// TwinCAT 3 PLC project main_program
// ProgramVersion: 3.1.4024.0
// libraries:
//   Tc2_MC2, * (Beckhoff Automation GmbH)
//   Tc2_Standard, * (Beckhoff Automation GmbH)
//   Tc2_System, * (Beckhoff Automation GmbH)
//   Tc3_Module, * (Beckhoff Automation GmbH)
// project tree:
//   DUTs/ E_BiaxialState.TcDUT (not stored), E_PlcSystemStatus.TcDUT (not stored), E_SafetyState.TcDUT (not stored), E_SyncPoint.TcDUT (not stored), ST_settings.TcDUT, ST_MoveCommand.TcDUT, ST_SystemStatus.TcDUT
//   GVLs/ GVL_Axis.TcGVL
//   / PlcTask.TcTTO
//   POUs/ fb_MovementController.TcPOU, fb_AxisStatusPublisher.TcPOU (not stored), fb_BiaxialCoordinator.TcPOU (not stored), fb_safety.TcPOU, fb_StatusBuffer.TcPOU, MAIN.TcPOU
// real-time tasks:
//   TASK PlcTask: cycle T#10ms, priority 20, ADS port 350
// motion (NC):
//   TASK NC-Task 1 SAF: cycle T#2ms, priority 4, ADS port 501
//   TASK NC-Task 1 SVB: cycle T#10ms, priority 8, ADS port 511
//   AXIS xAxis (id 1)
//     Dynamic: Acceleration=150, Deceleration=150, Jerk=225
//     Velo: RefSearch=2, RefSync=5, SlowManual=5, FastManual=10, Maximum=100
//     OtherSettings: AllowMotionCmdToSlave=true
//     encoder EncType=19
//       EncPara: ScaleFactorNumerator=2, ScaleFactorDenominator=1048576, MaxCount=#xffffffff
//         SoftEndMaxControl: Range=10000
//         Inc: RefSearchInverse=true, RefPosition=-5
//     drive DrvType=16
//       DrvPara: MaxCount=#xffffffff, DriveControlDWord=#x00020100
//         Analog: TorqueSetpointScale=10, ScaleFactorActTorque=0.1
//         TimeComp: TaskDelayCycles=1
//     controller CtrType=1
//       CtrPara: PriorControlFactor=1
//         Observer: BandWidth=20
//   AXIS yAxis (id 2)
//     Dynamic: Acceleration=150, Deceleration=150, Jerk=225
//     Velo: RefSearch=2, RefSync=5, SlowManual=5, FastManual=10, Maximum=100
//     OtherSettings: AllowMotionCmdToSlave=true
//     encoder EncType=19
//       EncPara: ScaleFactorNumerator=2, ScaleFactorDenominator=1048576, MaxCount=#xffffffff
//         SoftEndMinControl: Enable=true
//         SoftEndMaxControl: Range=10000
//         Inc: RefSearchInverse=true, RefPosition=-5, RefMode=1
//     drive DrvType=16
//       DrvPara: MaxCount=#xffffffff, DriveControlDWord=#x00020100
//         Analog: TorqueSetpointScale=10, ScaleFactorActTorque=0.1
//         TimeComp: TaskDelayCycles=1
//     controller CtrType=1
//       CtrPara: PriorControlFactor=1
//         Observer: BandWidth=20
// I/O:
//   DEVICE Device 1 (EtherCAT), AmsNetId 5.85.113.174.2.1
//     Term 1 (EK1200) [EK1200-5000 EtherCAT Power supply (2A E-Bus)]
//       Term 2 (EL7062) [EL7062-0000 2Ch. Stepper motor output stage (48V, 3A)]
//       Term 3 (EL9510) [EL9510 Power supply terminal 10V]
//       Term 4 (EL3356-0020) [EL3356-0020 1Ch. Ana. Input Resistor Bridge Terminal, 24bit, High Precision, with calibration certificate]
//       Term 5 (EL3356-0020) [EL3356-0020 1Ch. Ana. Input Resistor Bridge Terminal, 24bit, High Precision, with calibration certificate]
//       Term 6 (EL9011) [EL9011 End Terminal]
// variable links:
//   NC-Task 1 SAF/Axes/xAxis <-> Device 1 (EtherCAT)/Term 1 (EK1200)/Term 2 (EL7062)
//     Drive/Inputs/In/nDataIn1 <-> DRV Following error actual value Channel 2/Following error actual value
//     Drive/Inputs/In/nDcOutputTime <-> InfoData/DcOutputShift
//     Drive/Inputs/In/nState1 <-> DRV Statusword Channel 2/Statusword
//     Drive/Inputs/In/nState2 <-> DRV Statusword Channel 2/Statusword @bit 8
//     Drive/Inputs/In/nState4 @bit 1 <-> WcState/InputToggle
//     Drive/Inputs/In/nState4 <-> WcState/WcState
//     Drive/Outputs/Out/nCtrl1 <-> DRV Controlword Channel 2/Controlword
//     Drive/Outputs/Out/nCtrl2 <-> DRV Controlword Channel 2/Controlword @bit 8
//     Drive/Outputs/Out/nDataOut1 <-> DRV Target position Channel 2/Target position
//     Enc/Inputs/In/nDataIn1 <-> FB Position Channel 2/Position
//     Enc/Inputs/In/nDcInputTime <-> InfoData/DcInputShift
//     Enc/Inputs/In/nState4 @bit 1 <-> WcState/InputToggle
//     Enc/Inputs/In/nState4 <-> WcState/WcState
//   NC-Task 1 SAF/Axes/yAxis <-> Device 1 (EtherCAT)/Term 1 (EK1200)/Term 2 (EL7062)
//     Drive/Inputs/In/nDataIn1 <-> DRV Following error actual value Channel 1/Following error actual value
//     Drive/Inputs/In/nDcOutputTime <-> InfoData/DcOutputShift
//     Drive/Inputs/In/nState1 <-> DRV Statusword Channel 1/Statusword
//     Drive/Inputs/In/nState2 <-> DRV Statusword Channel 1/Statusword @bit 8
//     Drive/Inputs/In/nState4 @bit 1 <-> WcState/InputToggle
//     Drive/Inputs/In/nState4 <-> WcState/WcState
//     Drive/Outputs/Out/nCtrl1 <-> DRV Controlword Channel 1/Controlword
//     Drive/Outputs/Out/nCtrl2 <-> DRV Controlword Channel 1/Controlword @bit 8
//     Drive/Outputs/Out/nDataOut1 <-> DRV Target position Channel 1/Target position
//     Enc/Inputs/In/nDataIn1 <-> FB Position Channel 1/Position
//     Enc/Inputs/In/nDcInputTime <-> InfoData/DcInputShift
//     Enc/Inputs/In/nState4 @bit 1 <-> WcState/InputToggle
//     Enc/Inputs/In/nState4 <-> WcState/WcState
//   main program/main program Instance <-> Device 1 (EtherCAT)/Term 1 (EK1200)/Term 2 (EL7062)
//     PlcTask Inputs/MAIN.nEndStopHx <-> DI Inputs Channel 2/Input 1
//     PlcTask Inputs/MAIN.nEndStopHy <-> DI Inputs Channel 1/Input 2
//     PlcTask Inputs/MAIN.nEndStopLx <-> DI Inputs Channel 1/Input 1
//     PlcTask Inputs/MAIN.nEndStopLy <-> DI Inputs Channel 2/Input 2
//   main program/main program Instance <-> Device 1 (EtherCAT)/Term 1 (EK1200)/Term 4 (EL3356-0020)
//     PlcTask Inputs/MAIN.nRawTenzoX <-> RMB Value (INT32)/Value
//   main program/main program Instance <-> Device 1 (EtherCAT)/Term 1 (EK1200)/Term 5 (EL3356-0020)
//     PlcTask Inputs/MAIN.nRawTenzoY <-> RMB Value (INT32)/Value
//   main program/main program Instance <-> NC-Task 1 SAF/Axes/xAxis
//     PlcTask Inputs/GVL_Axis.xAxis.NcToPlc <-> Outputs/ToPlc
//     PlcTask Outputs/GVL_Axis.xAxis.PlcToNc <-> Inputs/FromPlc
//   main program/main program Instance <-> NC-Task 1 SAF/Axes/yAxis
//     PlcTask Inputs/GVL_Axis.yAxis.NcToPlc <-> Outputs/ToPlc
//     PlcTask Outputs/GVL_Axis.yAxis.PlcToNc <-> Inputs/FromPlc

CONFIGURATION main_program
    RESOURCE PLC ON TwinCAT3
        TASK PlcTask(INTERVAL := T#10ms, PRIORITY := 20);
        PROGRAM MAIN WITH PlcTask : MAIN;
    END_RESOURCE
END_CONFIGURATION

// ---- DUTs/ST_settings.TcDUT
TYPE ST_Settings :
	STRUCT
		// Force-sensor calibration
		fTenzoCons   : LREAL := 0.01;
		fTenzoOffset : LREAL := 0.0;

		// Force control
		fKp : LREAL := 10;
		fKi : LREAL := 0.1;
		fIntegralLimit  : LREAL := 10;
		fForceTolerance : LREAL := 0.1;
		fMaxVelocity    : LREAL := 100;

		// Runtime force limit
		fMaxForce            : LREAL := 10;
		fForceReliefDistance : LREAL := 1.0; // fixed overforce release move [mm]
		fForceReliefVelocity : LREAL := 1.0; // release speed [mm/s]
	END_STRUCT
END_TYPE

// ---- DUTs/ST_MoveCommand.TcDUT
TYPE ST_MoveCommand :
	STRUCT
		// Mode 1: one relative move
		fMoveDistance : LREAL;
		fMoveVelocity : LREAL;

		// Mode 2: one PI-regulated force hold
		fTargetForce   : LREAL;
		fForceDuration : LREAL;
	
		// Command and service controls
		nMode       : INT;  // 1=relative move, 2=force/time, 3=test sequence
		bExecute    : BOOL; // Start movement
		bHalt       : BOOL; // Panic stop
		bPower      : BOOL; // Maintained motor-enable request
		bReset      : BOOL; // Reset errors
		bHome       : BOOL; // Start homing sequence
		bStartTar   : BOOL; // Start tare sequence
		bSavePosition : BOOL; // Capture the current axis position while idle
		bRestorePosition : BOOL; // Return to the saved coordinate while idle
		fRestoreVelocity : LREAL; // Saved-position return speed [mm/s]

		// Optional force pre-conditioning sequence
		bIncludePreTest : BOOL;
		bPreTestOnly    : BOOL;  // Run pre-test and post-test without a main test
		nPreCycleCount  : INT;   // Number of force load/unload cycles, 0..50
		bPreloadEnabled : BOOL;  // Apply one force preload before the first cycle
		fPreloadValue   : LREAL; // Signed preload force [N]
		fPreCycleLoadValue : LREAL; // Signed repeated preconditioning load target [N]
		fPreUnloadValue : LREAL; // Signed force unload target [N]
		bPreUnloadToStart : BOOL; // Return to sequence-start position instead of force unload
		fPreTestRate     : LREAL; // Positive motor speed magnitude [mm/s]
		fPreTestForceTolerance : LREAL := 0.1; // Force deadband for pre-test endpoints [N]
		fPreloadHoldTime : LREAL := 0.0; // Hold time for the initial preload endpoint [s]
		fPreCycleHoldTime : LREAL := 0.0; // Hold time for cyclic pre-conditioning endpoints [s]

		// Main test settings
		fTestRate      : LREAL; // Positive motor speed magnitude [mm/s]
		fSingleForceTolerance : LREAL := 0.1; // Force deadband for single-test endpoints [N]
		fSingleForceHoldTime : LREAL := 0.0; // Hold time for the single-test primary force endpoint [s]
		fCyclicForceTolerance : LREAL := 0.1; // Force deadband for cyclic endpoints [N]
		fCyclicForceHoldTime : LREAL := 0.0; // Hold time for cyclic force endpoints [s]

		// Test selection: >0=cyclic count, 0=single test
		nCycleCount : INT;
		nLoadMode   : INT;   // 1=displacement, 2=force
		fLoadValues : ARRAY[1..50] OF LREAL; // per-cycle level [mm] or signed force [N]
		nUnloadMode : INT;   // 1=displacement, 2=force
		fUnloadValues : ARRAY[1..50] OF LREAL; // per-cycle level [mm] or signed force [N]

		// Single test (nMode=3, nCycleCount=0); criterion 2 is optional OR
		nStop1Mode         : INT;   // 0=off, 1=displacement, 2=force
		fStop1Value        : LREAL;
		nStop2Mode         : INT;
		fStop2Value        : LREAL;

		// 0=stay, 1=saved position, 2=sequence start,
		// 3=pre-test final position, 4=unload to zero force
		nPostTestMode : INT;
	END_STRUCT
END_TYPE

// ---- DUTs/ST_SystemStatus.TcDUT
TYPE ST_SystemStatus :
	STRUCT
		fPosBuffer   : ARRAY[1..50] OF LREAL; // FIFO position data
		fTenzoBuffer : ARRAY[1..50] OF LREAL; // FIFO tenzo data
		nBufferHead  : INT := 50;             // Index of latest completely written sample
		nSampleCounter    : UDINT := 0;       // Monotonic counter for dropped-sample detection
		nOperationCounter : UDINT := 0;       // Incremented after each completed motion command
		nInterfaceVersion : UDINT := 5;       // MATLAB/PLC ADS contract version
		fTenzoTarOffset   : LREAL := 0.0;     // Calculated tar offset
		fActPosition : LREAL := 0.0;          // Absolute NC axis position
		
		bWorking     : BOOL;                   // PLC occupied; do not send a new test
		bTarWorking  : BOOL;                   // PLC is calculating tare
		bError       : BOOL;                   // Latched application or motion error
		nErrorCode   : UDINT := 0;             // Application error code (0 = no error)
		nAxisErrorID : UDINT := 0;             // Native TwinCAT/NC error ID
		bPowered     : BOOL;                   // Axis power is enabled
		bHoming      : BOOL;                   // Homing command is active
		bHomed       : BOOL;                   // NC axis reports a valid home reference
		bStopped     : BOOL;                   // Axis is at standstill
		bSavedPositionValid : BOOL;            // A return-to-saved reference is available
		nTestPhase   : BYTE := 0;              // 0 idle, 1 pretest, 2 test, 3 post-test
	END_STRUCT
END_TYPE

// ---- GVLs/GVL_Axis.TcGVL
VAR_GLOBAL
	// Axis handlers
	xAxis : Axis_REF;
	yAxis : Axis_REF;
END_VAR

// ---- POUs/MAIN.TcPOU
PROGRAM MAIN

VAR
	fbSafetyX : fb_safety;
	fbSafetyY : fb_safety;
	fbSystemBufferX : fb_StatusBuffer;
	fbSystemBufferY : fb_StatusBuffer;
	fbMovementControllerX : fb_MovementController;
	fbMovementControllerY : fb_MovementController;
	fbBiaxialCoordinator : fb_BiaxialCoordinator;
	fbStatusPublisherX : fb_AxisStatusPublisher;
	fbStatusPublisherY : fb_AxisStatusPublisher;
	
	// DUTs import
	stMoveCommandX : ST_MoveCommand;
	stMoveCommandY : ST_MoveCommand;

	stSystemStatusX : ST_SystemStatus;
	stSystemStatusY : ST_SystemStatus;

	stSettingsX : ST_Settings;
	stSettingsY : ST_Settings;

	// IO Links
    nRawTenzoX AT %I* : DINT;
	nRawTenzoY AT %I* : DINT;

	nEndStopLx AT %I* : BOOL;
	nEndStopHx AT %I* : BOOL;

	nEndStopLy AT %I* : BOOL;
	nEndStopHy AT %I* : BOOL;

	// Normalized physical limits: TRUE means that the switch is pressed.
	bEndStopLxActive : BOOL;
	bEndStopHxActive : BOOL;
	bEndStopLyActive : BOOL;
	bEndStopHyActive : BOOL;

	// PLC-owned synchronized start request
	bStartBiaxialTest : BOOL; // ADS one-shot after both axis commands are prepared

END_VAR

VAR_TEMP
	bBiaxialAxesReady : BOOL;
	bBiaxialCommonAbortRequest : BOOL;
END_VAR

////////////////////////////////
//////////   safety   //////////
////////////////////////////////

// Refresh NC status before making any safety or motion decision
GVL_Axis.xAxis.ReadStatus();
GVL_Axis.yAxis.ReadStatus();

// Normalize the active-low physical switches
bEndStopLxActive := NOT nEndStopLx;
bEndStopHxActive := NOT nEndStopHx;
bEndStopLyActive := NOT nEndStopLy;
bEndStopHyActive := NOT nEndStopHy;

fbSafetyX(
    stAxis := GVL_Axis.xAxis,
    bPower := stMoveCommandX.bPower,
    bReset := stMoveCommandX.bReset,
    bHalt := stMoveCommandX.bHalt OR fbMovementControllerX.stateHalt,
    bHome := stMoveCommandX.bHome,
    bEndStopL := bEndStopLxActive,
	bEndStopH := bEndStopHxActive,
	bExternalBusy := fbMovementControllerX.bBusy OR stSystemStatusX.bTarWorking
);

fbSafetyY(
    stAxis := GVL_Axis.yAxis,
    bPower := stMoveCommandY.bPower,
    bReset := stMoveCommandY.bReset,
    bHalt := stMoveCommandY.bHalt OR fbMovementControllerY.stateHalt,
    bHome := stMoveCommandY.bHome,
	bEndStopL := bEndStopLyActive,
	bEndStopH := bEndStopHyActive,
	bExternalBusy := fbMovementControllerY.bBusy OR stSystemStatusY.bTarWorking
);

////////////////////////////////
////////// Update data /////////
////////////////////////////////

fbSystemBufferX(
	stSystemStatus:= stSystemStatusX,
	bBlockTar:= fbMovementControllerX.bBusy OR fbSafetyX.bHoming,
	nRawTenzo:= nRawTenzoX,
	fTenzoCons:=stSettingsX.fTenzoCons,
	fTenzoOffset:= stSettingsX.fTenzoOffset,
	bStartTar:= stMoveCommandX.bStartTar,
	fActPosition:= GVL_Axis.xAxis.NcToPlc.ActPos);
	
fbSystemBufferY(
	stSystemStatus:= stSystemStatusY,
	bBlockTar:= fbMovementControllerY.bBusy OR fbSafetyY.bHoming,
	nRawTenzo:= nRawTenzoY,
	fTenzoCons:=stSettingsY.fTenzoCons,
	fTenzoOffset:= stSettingsY.fTenzoOffset,
	bStartTar:= stMoveCommandY.bStartTar,
	fActPosition:= GVL_Axis.yAxis.NcToPlc.ActPos);

/////////////////////////////////////
////////// Main Move Logic //////////
/////////////////////////////////////

// A shared request starts both axes in one PLC scan. Single-axis tests keep
// using their individual bExecute fields and never enable synchronization.
bBiaxialAxesReady :=
	NOT fbMovementControllerX.bBusy AND
	NOT fbMovementControllerY.bBusy AND
	NOT fbMovementControllerX.bError AND
	NOT fbMovementControllerY.bError AND
	NOT fbSafetyX.bError AND NOT fbSafetyY.bError AND
	NOT fbSafetyX.bHoming AND NOT fbSafetyY.bHoming AND
	NOT stSystemStatusX.bTarWorking AND
	NOT stSystemStatusY.bTarWorking AND
	fbSafetyX.bPowerStatus AND fbSafetyY.bPowerStatus;

// Ignore ProtectiveStop when it was produced by the controller's own
// controlled halt. Operator, end-stop and independent safety stops abort both
// axes; an overforce relief request aborts only the synchronized peer.
bBiaxialCommonAbortRequest :=
	fbMovementControllerX.bError OR fbMovementControllerY.bError OR
	fbSafetyX.bError OR fbSafetyY.bError OR
	(fbSafetyX.bProtectiveStop AND
	 NOT fbMovementControllerX.stateHalt) OR
	(fbSafetyY.bProtectiveStop AND
	 NOT fbMovementControllerY.stateHalt) OR
	(bEndStopLxActive AND GVL_Axis.xAxis.Status.NegativeDirection) OR
	(bEndStopHxActive AND GVL_Axis.xAxis.Status.PositiveDirection) OR
	(bEndStopLyActive AND GVL_Axis.yAxis.Status.NegativeDirection) OR
	(bEndStopHyActive AND GVL_Axis.yAxis.Status.PositiveDirection) OR
	stMoveCommandX.bHalt OR stMoveCommandY.bHalt;

fbBiaxialCoordinator(
	bStartRequest := bStartBiaxialTest,
	bResetRequest := stMoveCommandX.bReset OR stMoveCommandY.bReset,
	bAxesReady := bBiaxialAxesReady,
	bCommonAbortRequest := bBiaxialCommonAbortRequest,
	bBusyX := fbMovementControllerX.bBusy,
	bBusyY := fbMovementControllerY.bBusy,
	bSavedPositionValidX := fbMovementControllerX.bSavedPositionValid,
	bSavedPositionValidY := fbMovementControllerY.bSavedPositionValid,
	nSyncPointX := fbMovementControllerX.nSyncPoint,
	nSyncPointY := fbMovementControllerY.nSyncPoint,
	nSyncCycleX := fbMovementControllerX.nSyncCycle,
	nSyncCycleY := fbMovementControllerY.nSyncCycle,
	bPeerAbortRequestX := fbMovementControllerX.bPeerAbortRequest,
	bPeerAbortRequestY := fbMovementControllerY.bPeerAbortRequest,
	stCommandX := stMoveCommandX,
	stCommandY := stMoveCommandY);

IF bStartBiaxialTest THEN
	bStartBiaxialTest := FALSE;
END_IF

IF fbBiaxialCoordinator.bStartBoth THEN
	stMoveCommandX.bExecute := TRUE;
	stMoveCommandY.bExecute := TRUE;
END_IF

fbMovementControllerX(
	Axis := GVL_Axis.xAxis,
	stMoveCommand := stMoveCommandX,
	stSettings := stSettingsX,
	fActPosition := GVL_Axis.xAxis.NcToPlc.ActPos,
    bPowerState := fbSafetyX.bPowerStatus,
	bHaltDone := fbSafetyX.bHaltDone,
	bSafetyError := fbSafetyX.bError,
	bProtectiveStop := fbSafetyX.bProtectiveStop,
	bExternalBusy := fbSafetyX.bHoming OR stSystemStatusX.bTarWorking,
	bSyncEnabled := fbBiaxialCoordinator.bSyncActive,
	bSyncRelease := fbBiaxialCoordinator.bSyncRelease,
	bSyncAbort := fbBiaxialCoordinator.bAbortX,
    fForce := stSystemStatusX.fTenzoBuffer[stSystemStatusX.nBufferHead]);

fbMovementControllerY(
	Axis := GVL_Axis.yAxis,
	stMoveCommand := stMoveCommandY,
	stSettings := stSettingsY,
	fActPosition := GVL_Axis.yAxis.NcToPlc.ActPos,
    bPowerState := fbSafetyY.bPowerStatus,
	bHaltDone := fbSafetyY.bHaltDone,
	bSafetyError := fbSafetyY.bError,
	bProtectiveStop := fbSafetyY.bProtectiveStop,
	bExternalBusy := fbSafetyY.bHoming OR stSystemStatusY.bTarWorking,
	bSyncEnabled := fbBiaxialCoordinator.bSyncActive,
	bSyncRelease := fbBiaxialCoordinator.bSyncRelease,
	bSyncAbort := fbBiaxialCoordinator.bAbortY,
	fForce := stSystemStatusY.fTenzoBuffer[stSystemStatusY.nBufferHead]);

///////////////////////////////////////////////////
////// ADS status contract for each axis //////////
///////////////////////////////////////////////////

fbStatusPublisherX(
	fActPosition := GVL_Axis.xAxis.NcToPlc.ActPos,
	bPowerStatus := fbSafetyX.bPowerStatus,
	bHoming := fbSafetyX.bHoming,
	bHomed := fbSafetyX.bHomed,
	bStopped := fbSafetyX.bStopped,
	bProtectiveStop := fbSafetyX.bProtectiveStop,
	bSafetyError := fbSafetyX.bError,
	nSafetyErrorCode := fbSafetyX.nErrorCode,
	nSafetyAxisErrorID := fbSafetyX.nAxisErrorID,
	bMovementBusy := fbMovementControllerX.bBusy,
	bMovementError := fbMovementControllerX.bError,
	nMovementStatus := fbMovementControllerX.nSystemStatus,
	nMovementErrorCode := fbMovementControllerX.nErrorCode,
	nMovementAxisErrorID := fbMovementControllerX.nAxisErrorID,
	nOperationCounter := fbMovementControllerX.nOperationCounter,
	bSavedPositionValid := fbMovementControllerX.bSavedPositionValid,
	bStartError := fbBiaxialCoordinator.bStartError,
	nStartErrorCode := fbBiaxialCoordinator.nStartErrorCode,
	stSystemStatus := stSystemStatusX);

fbStatusPublisherY(
	fActPosition := GVL_Axis.yAxis.NcToPlc.ActPos,
	bPowerStatus := fbSafetyY.bPowerStatus,
	bHoming := fbSafetyY.bHoming,
	bHomed := fbSafetyY.bHomed,
	bStopped := fbSafetyY.bStopped,
	bProtectiveStop := fbSafetyY.bProtectiveStop,
	bSafetyError := fbSafetyY.bError,
	nSafetyErrorCode := fbSafetyY.nErrorCode,
	nSafetyAxisErrorID := fbSafetyY.nAxisErrorID,
	bMovementBusy := fbMovementControllerY.bBusy,
	bMovementError := fbMovementControllerY.bError,
	nMovementStatus := fbMovementControllerY.nSystemStatus,
	nMovementErrorCode := fbMovementControllerY.nErrorCode,
	nMovementAxisErrorID := fbMovementControllerY.nAxisErrorID,
	nOperationCounter := fbMovementControllerY.nOperationCounter,
	bSavedPositionValid := fbMovementControllerY.bSavedPositionValid,
	bStartError := fbBiaxialCoordinator.bStartError,
	nStartErrorCode := fbBiaxialCoordinator.nStartErrorCode,
	stSystemStatus := stSystemStatusY);

// Home and reset are one-shot commands
stMoveCommandX.bHome := FALSE;
stMoveCommandY.bHome := FALSE;
stMoveCommandX.bReset := FALSE;
stMoveCommandY.bReset := FALSE;
stMoveCommandX.bSavePosition := FALSE;
stMoveCommandY.bSavePosition := FALSE;
stMoveCommandX.bRestorePosition := FALSE;
stMoveCommandY.bRestorePosition := FALSE;

END_PROGRAM

// ---- POUs/fb_safety.TcPOU
FUNCTION_BLOCK fb_safety
VAR_INPUT
	bPower        : BOOL;
	bReset        : BOOL;
	bHalt         : BOOL;
	bHome         : BOOL;
	bEndStopL     : BOOL; // TRUE when the normalized lower switch is active
	bEndStopH     : BOOL; // TRUE when the normalized upper switch is active
	bExternalBusy : BOOL; // Test motion or tare is active
END_VAR

VAR_OUTPUT
	bPowerStatus       : BOOL;
	bHaltDone          : BOOL;
	bError             : BOOL;
	nErrorCode         : UDINT;
	nAxisErrorID       : UDINT;
	bHoming            : BOOL;
	bHomed             : BOOL;
	bStopped           : BOOL;
	bProtectiveStop    : BOOL; // Abort active test motion but retain commanded power
END_VAR

VAR_IN_OUT
	stAxis : AXIS_REF;
END_VAR

VAR
	fbPower        : MC_Power;
	fbReset        : MC_Reset;
	fbHalt         : MC_Halt;
	fbHome         : MC_Home;
	fbMoveToZero   : MC_MoveRelative;

	rtReset        : R_TRIG;
	rtHalt         : R_TRIG;
	rtHome         : R_TRIG;

	fbHomeTimeout  : TON;
	fbMoveTimeout  : TON;

	eState             : E_SafetyState := E_SafetyState.Idle;
	bFaultPowerInhibit : BOOL;
	bResetExecute      : BOOL;
	bHaltDonePulse     : BOOL;
	fHomeParkDistance  : LREAL;
END_VAR

VAR CONSTANT
	HOME_PARK_POSITION : LREAL := 0.0;
	HOME_PARK_VELOCITY : LREAL := 5.0;
	HOME_TIMEOUT       : TIME := T#10M;
	HOME_PARK_TIMEOUT  : TIME := T#10S;
END_VAR


// Commands are edge-triggered
rtReset(CLK := bReset);
rtHalt(CLK := bHalt);
rtHome(CLK := bHome);

// halt pulse is one cicle variable
bHaltDonePulse := FALSE;

// Reset a latched fault
IF rtReset.Q AND bError AND eState = E_SafetyState.Idle THEN
	bResetExecute := TRUE;
END_IF

IF bResetExecute AND fbReset.Done THEN
	bResetExecute := FALSE;
	bError := FALSE;
	nErrorCode := 0;
	nAxisErrorID := 0;
	bFaultPowerInhibit := FALSE;
ELSIF bResetExecute AND fbReset.Error THEN
	bResetExecute := FALSE;
	bError := TRUE;
	nErrorCode := 1002;
	nAxisErrorID := fbReset.ErrorID;
	bFaultPowerInhibit := TRUE;
END_IF

// Latch genuine NC, wiring and motion-function-block faults
IF NOT bError THEN
	IF stAxis.Status.Error THEN
		bError := TRUE;
		nErrorCode := 1005;
		nAxisErrorID := stAxis.Status.ErrorID;
		eState := E_SafetyState.ErrorStop;
	ELSIF bEndStopL AND bEndStopH THEN
		bError := TRUE;
		nErrorCode := 1006;
		nAxisErrorID := 0;
		eState := E_SafetyState.ErrorStop;
	ELSIF fbPower.Error THEN
		bError := TRUE;
		nErrorCode := 1001;
		nAxisErrorID := fbPower.ErrorID;
		eState := E_SafetyState.ErrorStop;
	ELSIF fbHalt.Error THEN
		bError := TRUE;
		nErrorCode := 1003;
		nAxisErrorID := fbHalt.ErrorID;
		eState := E_SafetyState.ErrorStop;
	ELSIF fbHome.Error THEN
		bError := TRUE;
		nErrorCode := 1004;
		nAxisErrorID := fbHome.ErrorID;
		eState := E_SafetyState.ErrorStop;
	ELSIF fbMoveToZero.Error THEN
		bError := TRUE;
		nErrorCode := 1008;
		nAxisErrorID := fbMoveToZero.ErrorID;
		eState := E_SafetyState.ErrorStop;
	END_IF
END_IF

// Halt and switch to error stop
IF rtHalt.Q AND eState <> E_SafetyState.ErrorStop THEN
	eState := E_SafetyState.ProtectiveStop;
END_IF

CASE eState OF
	E_SafetyState.Idle:
		// Stop only when travelling farther into an active physical switch.
		IF (bEndStopL AND stAxis.Status.NegativeDirection) OR
			(bEndStopH AND stAxis.Status.PositiveDirection) THEN
			eState := E_SafetyState.ProtectiveStop;
		ELSIF rtHome.Q AND NOT bExternalBusy AND fbPower.Status THEN
			eState := E_SafetyState.Homing;
		END_IF

	E_SafetyState.Homing:
		IF fbHomeTimeout.Q THEN
			bError := TRUE;
			nErrorCode := 1011;
			nAxisErrorID := 0;
			eState := E_SafetyState.ErrorStop;
		ELSIF fbHome.Done THEN
			IF bEndStopL THEN
				bError := TRUE;
				nErrorCode := 1014;
				nAxisErrorID := 0;
				eState := E_SafetyState.ErrorStop;
			ELSE
				fHomeParkDistance := HOME_PARK_POSITION - stAxis.NcToPlc.ActPos;
				eState := E_SafetyState.MoveToZero;
			END_IF
		END_IF

	E_SafetyState.MoveToZero:
		IF bEndStopH THEN
			bError := TRUE;
			nErrorCode := 1013;
			nAxisErrorID := 0;
			eState := E_SafetyState.ErrorStop;
		ELSIF fbMoveTimeout.Q THEN
			bError := TRUE;
			nErrorCode := 1012;
			nAxisErrorID := 0;
			eState := E_SafetyState.ErrorStop;
		ELSIF fbMoveToZero.Done THEN
			eState := E_SafetyState.Complete;
		END_IF

	E_SafetyState.Complete:
		eState := E_SafetyState.Idle;

	E_SafetyState.ProtectiveStop:
		IF fbHalt.Done OR stAxis.Status.StandStill THEN
			bHaltDonePulse := TRUE;
			eState := E_SafetyState.Idle;
		END_IF

	E_SafetyState.ErrorStop:
		IF fbHalt.Done OR stAxis.Status.StandStill THEN
			bHaltDonePulse := TRUE;
			bFaultPowerInhibit := TRUE;
			eState := E_SafetyState.Idle;
		END_IF
END_CASE

fbHomeTimeout(
	IN := eState = E_SafetyState.Homing,
	PT := HOME_TIMEOUT);
fbMoveTimeout(
	IN := eState = E_SafetyState.MoveToZero,
	PT := HOME_PARK_TIMEOUT);

// Physical switches continuously block motion farther into the active limit
fbPower(
	Axis := stAxis,
	Enable := bPower AND NOT bFaultPowerInhibit,
	Enable_Positive := bPower AND NOT bFaultPowerInhibit AND NOT bEndStopH,
	Enable_Negative := bPower AND NOT bFaultPowerInhibit AND (NOT bEndStopL OR eState = E_SafetyState.Homing),
	Override := 100.0);

fbReset(
	Axis := stAxis,
	Execute := bResetExecute);

// TwinCAT NC owns the complete reference-cam search and release sequence.
// Position is omitted so the NC-configured reference position (-5 mm) is used.
fbHome(
	Axis := stAxis,
	Execute := eState = E_SafetyState.Homing,
	HomingMode := MC_DefaultHoming,
	BufferMode := MC_Aborting,
	bCalibrationCam := bEndStopL);

// Park at the safe working origin after TwinCAT has established the reference.
fbMoveToZero(
	Axis := stAxis,
	Execute := eState = E_SafetyState.MoveToZero,
	Distance := fHomeParkDistance,
	Velocity := HOME_PARK_VELOCITY,
	BufferMode := MC_Aborting);

fbHalt(
	Axis := stAxis,
	Execute := eState = E_SafetyState.ProtectiveStop OR
		eState = E_SafetyState.ErrorStop);

// Public status.
bPowerStatus := fbPower.Status;
bHaltDone := bHaltDonePulse OR fbHalt.Done;
bHoming := eState = E_SafetyState.Homing OR
	eState = E_SafetyState.MoveToZero;
bHomed := stAxis.Status.Homed;
bStopped := stAxis.Status.StandStill;
bProtectiveStop := eState = E_SafetyState.ProtectiveStop;

END_FUNCTION_BLOCK

// ---- POUs/fb_StatusBuffer.TcPOU
FUNCTION_BLOCK fb_StatusBuffer
VAR_IN_OUT
    stSystemStatus    : ST_SystemStatus;
    bStartTar         : BOOL;  // Cleared after completion or when tare is blocked
END_VAR
VAR_INPUT
	bBlockTar     : BOOL;  // Motion or homing is active

	// Tenzo buffer
    nRawTenzo    : DINT;
    fTenzoCons   : LREAL;
    fTenzoOffset : LREAL;
	
	// Position buffer
	fActPosition   : LREAL;
	fStartPosition : LREAL;
END_VAR
VAR
    fbStartTarRiseClp : R_TRIG;   // Detects the moment tare button is pressed
    bTarActive        : BOOL;     // Flag indicating taring is in progress
    nTarCounter       : INT;      // Counts up to 100 samples
    fTarAccumulator   : LREAL;    // Holds the running sum of samples
    fCurrentCalculated: LREAL;    // The current weight before tare constant
	nNextHead        : INT;
END_VAR


// Calculate the current weight snapshot
fCurrentCalculated := (DINT_TO_LREAL(nRawTenzo) * fTenzoCons) + fTenzoOffset;

// Taring Logic
// Reject a tare command received while motion or homing is active.
IF bStartTar AND bBlockTar THEN
	bStartTar := FALSE;
END_IF

fbStartTarRiseClp(CLK := bStartTar);

// Start the taring process
IF fbStartTarRiseClp.Q AND NOT bTarActive THEN
    bTarActive      := TRUE;
    nTarCounter     := 0;
    fTarAccumulator := 0.0;
END_IF

IF bTarActive THEN
    // Accumulate the current weight across 100 consecutive cycles
    fTarAccumulator := fTarAccumulator + fCurrentCalculated;
    nTarCounter     := nTarCounter + 1;
    
    // After 100 
    IF nTarCounter >= 100 THEN
        // Calculate the mean
        stSystemStatus.fTenzoTarOffset := - (fTarAccumulator / 100.0); 
        
        // Reset control flags
        bTarActive := FALSE;
        bStartTar  := FALSE;
    END_IF
END_IF

// Flag sys is working so no mowement will be done
stSystemStatus.bTarWorking := bTarActive;

// New head
nNextHead := stSystemStatus.nBufferHead + 1;
IF nNextHead > 50 THEN
    nNextHead := 1;
END_IF

// Buffering data
stSystemStatus.fTenzoBuffer[nNextHead] := fCurrentCalculated + stSystemStatus.fTenzoTarOffset;
stSystemStatus.fPosBuffer[nNextHead] := fActPosition - fStartPosition;

// Matlab status helpers
stSystemStatus.nBufferHead := nNextHead;
stSystemStatus.nSampleCounter := stSystemStatus.nSampleCounter + 1;

END_FUNCTION_BLOCK

// ---- POUs/fb_MovementController.TcPOU
FUNCTION_BLOCK fb_MovementController
VAR_INPUT
	fForce        : LREAL; // Actual force
	fActPosition  : LREAL; // Absolute NC position
	bPowerState   : BOOL;  // Actual power on state
	bHaltDone     : BOOL;  // Motor stopped
	bSafetyError  : BOOL;
	bProtectiveStop : BOOL;
	bExternalBusy : BOOL;
	bSyncEnabled  : BOOL;  // TRUE only for a PLC-owned biaxial test
	bSyncRelease  : BOOL;  // Shared barrier release from MAIN
	bSyncAbort    : BOOL;  // Stop this axis when the synchronized peer aborts
	stSettings    : ST_Settings;
END_VAR

VAR_OUTPUT
	fTestStartPos : LREAL := 0.0; // position where test started
	stateHalt   : BOOL; // Request a controlled stop
	bBusy       : BOOL; // System is processing a test or stopping
	bError      : BOOL; // Latched application/motion error
	nErrorCode  : UDINT;
	nAxisErrorID: UDINT;
	nOperationCounter : UDINT;
	bSavedPositionValid : BOOL;
	nSystemStatus : INT; // High-level numeric system status exposed through ADS
	nSyncPoint : BYTE; // E_SyncPoint: 0 none through 6 pretension
	nSyncCycle : INT;  // Cycle associated with the current sync point
	bPeerAbortRequest : BOOL; // Abort synchronized peer while local relief continues
END_VAR

VAR
	// Movement FBs
	fbMC_MoveRelative1 : MC_MoveRelative;
	fbMC_MoveVelocity  : MC_MoveVelocity;
	
	// Shared help vars
	nSeqState    : INT; // Current sequence state
	
	// mode 1
	fTargetDist1 : LREAL;
	fTargetVel1  : LREAL;
	
	// mode 2/3 vel movement
	bExecuteVelMove : BOOL;
    fCmdVelocity    : LREAL;
    mcDirection     : MC_Direction;
	
	// mode 2/3 help vars
	fTargetForce          : LREAL; // Wanted F
    fForceError           : LREAL; // Regulation error
    fForceErrorIntegral   : LREAL; // Integ of error
	fMode2HoldElapsed     : LREAL; // Accumulated time inside force tolerance
	fLastSentVelocity   : LREAL;    // Tracks last updated velocity to prevent NC spamming
	fPendingVelocity   : LREAL;
	mcPendingDirection : MC_Direction;
	nVelocityState     : INT;
	nVelocityUpdateCounter : INT;
	bResetRequested : BOOL;
	bOperationCompleted : BOOL;

	// Saved/reference positions
	fSavedPosition      : LREAL;
	fPreTestFinalPos    : LREAL;
	rtSavePosition      : R_TRIG;
	rtRestorePosition   : R_TRIG;
	rtSyncAbort         : R_TRIG;

	// Generic endpoint engine for test-sequence mode 3
	nCurrentCycle           : INT;
	nCurrentPreCycle        : INT;
	nAfterEndpointState     : INT;
	fEndpointTargetPosition : LREAL;
	fEndpointTargetForce    : LREAL;
	fEndpointRate           : LREAL;
	fEndpointTolerance      : LREAL;
	fEndpointHoldTime       : LREAL;
	fEndpointStartError     : LREAL;
	fEndpointCurrentError   : LREAL;
	fForceHoldElapsed       : LREAL;
	nLoadDirection          : INT;
	nLastMotionDirection    : INT;
	nReliefSourceDirection  : INT;
	nEndpointSyncPoint      : BYTE;
	nEndpointSyncCycle      : INT;
	bForceEndpointReady     : BOOL;

	// Optional OR criterion for the single test
	bSinglePrimaryActive  : BOOL;
	bSingleStopReached    : BOOL;
	fStop2TargetPosition  : LREAL;
	fStop2StartError      : LREAL;
	fStop2CurrentError    : LREAL;
	
END_VAR

VAR CONSTANT
	// Task and controller constants
	CYCLE_TIME : LREAL := 0.01; // dt of plc
	VELOCITY_UPDATE_DELTA : LREAL := 0.1;
	VELOCITY_UPDATE_CYCLES : INT := 10;
	POSITION_EPSILON : LREAL := 0.000001;
	FORCE_POLARITY : INT := -1;
	STATUS_IDLE : INT := 0;
	STATUS_STOPPING : INT := 3;
	STATUS_BASIC_MOVE : INT := 5;
	STATUS_FORCE_MODE : INT := 6;
	STATUS_PRETENSION : INT := 10;
	STATUS_PRETEST_CYCLIC : INT := 11;
	STATUS_SINGLE_TEST : INT := 20;
	STATUS_CYCLIC_TEST : INT := 21;
	STATUS_POSTTEST : INT := 30;
	SYNC_NONE : BYTE := 0;
	SYNC_PRETEST_DONE : BYTE := 1;
	SYNC_LOAD_DONE : BYTE := 2;
	SYNC_UNLOAD_DONE : BYTE := 3;
	SYNC_MAIN_DONE : BYTE := 4;
	SYNC_POSTTEST_DONE : BYTE := 5;
	SYNC_PRETENSION_DONE : BYTE := 6;
	STATE_IDLE : INT := 0;
	STATE_MODE_START : INT := 1;
	STATE_MODE_RUN : INT := 2;
	STATE_PRELOAD : INT := 10;
	STATE_CAPTURE_TEST_START : INT := 11;
	STATE_PRE_CYCLE_LOAD : INT := 12;
	STATE_PRE_CYCLE_UNLOAD : INT := 13;
	STATE_PRE_CYCLE_NEXT : INT := 14;
	STATE_CAPTURE_PRETEST_FINAL : INT := 18;
	STATE_PRETEST_BARRIER : INT := 19;
	STATE_SELECT_MAIN_TEST : INT := 20;
	STATE_SECONDARY_BARRIER : INT := 49;
	STATE_POSTTEST_SELECT : INT := 50;
	STATE_POSTTEST_WAIT_STOP : INT := 51;
	STATE_POSTTEST_BARRIER : INT := 54;
	STATE_OPERATION_COMPLETE : INT := 55;
	STATE_RESTORE_COMPLETE : INT := 56;
	STATE_CYCLIC_LOAD : INT := 100;
	STATE_CYCLIC_UNLOAD : INT := 110;
	STATE_CYCLIC_NEXT : INT := 120;
	STATE_CYCLIC_COMPLETE : INT := 121;
	STATE_SINGLE_START : INT := 200;
	STATE_SINGLE_WAIT_STOP : INT := 220;
	STATE_POSITION_PREPARE : INT := 300;
	STATE_POSITION_EXECUTE : INT := 301;
	STATE_POSITION_WAIT : INT := 302;
	STATE_POSITION_BARRIER : INT := 303;
	STATE_FORCE_PREPARE : INT := 310;
	STATE_FORCE_EXECUTE : INT := 311;
	STATE_FORCE_WAIT_TOLERANCE : INT := 312;
	STATE_FORCE_WAIT_STOP : INT := 313;
	STATE_FORCE_HOLD : INT := 314;
	STATE_ABORT_STOPPING : INT := 900;
	STATE_RELIEF_WAIT_STOP : INT := 910;
	STATE_RELIEF_START : INT := 911;
	STATE_RELIEF_WAIT_MOVE : INT := 912;
	STATE_ERROR_STOPPING : INT := 998;
	STATE_ERROR_LATCHED : INT := 999;
	ERROR_UNSUPPORTED_MODE : UDINT := 2001;
	ERROR_SAVED_POSITION_UNAVAILABLE : UDINT := 2002;
	ERROR_UNSUPPORTED_ENDPOINT : UDINT := 2003;
	ERROR_UNSUPPORTED_POST_ACTION : UDINT := 2005;
	ERROR_POWER_UNAVAILABLE : UDINT := 2006;
	ERROR_INVALID_CONFIGURATION : UDINT := 2007;
	ERROR_COMMAND_CONFLICT : UDINT := 2008;
	ERROR_INVALID_RUNTIME_VALUE : UDINT := 2009;
	ERROR_RELIEF_COMPLETED : UDINT := 2101;
	ERROR_RELIEF_DIRECTION_UNKNOWN : UDINT := 2102;
	ERROR_RELATIVE_MOVE : UDINT := 2201;
	ERROR_VELOCITY_MOVE : UDINT := 2203;
END_VAR

VAR_IN_OUT
	Axis          : AXIS_REF;
	stMoveCommand : ST_MoveCommand;
END_VAR


// =========================================================
//                    Saved position
// =========================================================

rtSavePosition(CLK := stMoveCommand.bSavePosition);
rtRestorePosition(CLK := stMoveCommand.bRestorePosition);
rtSyncAbort(CLK := bSyncEnabled AND bSyncAbort);
IF rtSavePosition.Q AND nSeqState = STATE_IDLE AND NOT bExternalBusy THEN
	fSavedPosition := fActPosition;
	bSavedPositionValid := TRUE;
END_IF

// =========================================================
//                      Error handling
// =========================================================

IF stMoveCommand.bReset THEN
	bResetRequested := TRUE;
END_IF

IF bResetRequested AND bError AND NOT bSafetyError THEN
	bError := FALSE;
	nErrorCode := 0;
	nAxisErrorID := 0;
	nSeqState := STATE_IDLE;
	stateHalt := FALSE;
	bResetRequested := FALSE;
ELSIF bResetRequested AND NOT bError AND NOT bSafetyError THEN
	IF nSeqState = STATE_ERROR_LATCHED THEN
		nSeqState := STATE_IDLE;
	END_IF
	bResetRequested := FALSE;
END_IF

// Operator and safety stops abort the sequence without running post-test.
IF stMoveCommand.bHalt OR (bProtectiveStop AND NOT stateHalt) OR
	rtSyncAbort.Q THEN
	IF stMoveCommand.bHalt THEN
		stMoveCommand.bHalt := FALSE;
	END_IF
	stMoveCommand.bExecute := FALSE;
	ClearActiveCommand();
	stateHalt := TRUE;
	nSeqState := STATE_ABORT_STOPPING;
END_IF

// A safety-owned error cancels local motion without issuing another halt.
IF bSafetyError THEN
	stMoveCommand.bExecute := FALSE;
	ClearActiveCommand();
	stateHalt := FALSE;
	nSeqState := STATE_ERROR_LATCHED;
END_IF

// Latch motion-function-block and sensor errors.
IF NOT bError AND NOT bSafetyError THEN
	IF fbMC_MoveRelative1.Error THEN
		bError := TRUE;
		nErrorCode := ERROR_RELATIVE_MOVE;
		nAxisErrorID := fbMC_MoveRelative1.ErrorID;
	ELSIF fbMC_MoveVelocity.Error THEN
		bError := TRUE;
		nErrorCode := ERROR_VELOCITY_MOVE;
		nAxisErrorID := fbMC_MoveVelocity.ErrorID;
	ELSIF nSeqState > STATE_IDLE AND
		nSeqState < STATE_ABORT_STOPPING AND
		NOT ((fForce = fForce) AND ABS(fForce) < 1.0E300) THEN
		bError := TRUE;
		nErrorCode := ERROR_INVALID_RUNTIME_VALUE;
	END_IF
END_IF

// Runtime overforce response: halt, make one fixed relative release move, then abort.
IF NOT bError AND NOT bSafetyError AND
	nSeqState > STATE_IDLE AND nSeqState < STATE_ABORT_STOPPING AND
	ABS(fForce) > stSettings.fMaxForce THEN
	IF stMoveCommand.nMode = 3 AND nLoadDirection <> 0 THEN
		nReliefSourceDirection := nLoadDirection;
	ELSIF Axis.Status.PositiveDirection THEN
		nReliefSourceDirection := 1;
	ELSIF Axis.Status.NegativeDirection THEN
		nReliefSourceDirection := -1;
	ELSE
		nReliefSourceDirection := nLastMotionDirection;
	END_IF
	fbMC_MoveRelative1.Execute := FALSE;
	bExecuteVelMove := FALSE;
	bSinglePrimaryActive := FALSE;
	bForceEndpointReady := FALSE;
	nSyncPoint := SYNC_NONE;
	nSyncCycle := 0;
	stateHalt := TRUE;
	nSeqState := STATE_RELIEF_WAIT_STOP;
END_IF

IF bError AND nSeqState <> STATE_ERROR_STOPPING AND
	nSeqState <> STATE_ERROR_LATCHED THEN
	stMoveCommand.bExecute := FALSE;
	ClearActiveCommand();
	stateHalt := TRUE;
	nSeqState := STATE_ERROR_STOPPING;
END_IF

IF bError THEN
	stMoveCommand.bExecute := FALSE;
END_IF

IF stMoveCommand.bExecute AND bExternalBusy THEN
	stMoveCommand.bExecute := FALSE;
	bError := TRUE;
	nErrorCode := ERROR_COMMAND_CONFLICT;
END_IF

IF stMoveCommand.bExecute AND NOT bPowerState THEN
	stMoveCommand.bExecute := FALSE;
	bError := TRUE;
	nErrorCode := ERROR_POWER_UNAVAILABLE;
END_IF

// Finish operator/error stops.
IF (nSeqState = STATE_ABORT_STOPPING OR
	nSeqState = STATE_ERROR_STOPPING) AND bHaltDone THEN
	stateHalt := FALSE;
	IF nSeqState = STATE_ERROR_STOPPING THEN
		nSeqState := STATE_ERROR_LATCHED;
	ELSE
		nSeqState := STATE_IDLE;
	END_IF
END_IF

// Overforce release sequence. FB1 is reused with aborting buffer mode.
CASE nSeqState OF
	STATE_RELIEF_WAIT_STOP:
		IF bHaltDone THEN
			stateHalt := FALSE;
			IF nReliefSourceDirection = 0 THEN
				bError := TRUE;
				nErrorCode := ERROR_RELIEF_DIRECTION_UNKNOWN;
				nSeqState := STATE_ERROR_LATCHED;
			ELSE
				fTargetDist1 := -INT_TO_LREAL(nReliefSourceDirection) *
					ABS(stSettings.fForceReliefDistance);
				fTargetVel1 := ABS(stSettings.fForceReliefVelocity);
				fbMC_MoveRelative1.Execute := FALSE;
				nSeqState := STATE_RELIEF_START;
			END_IF
		END_IF

	STATE_RELIEF_START:
		fbMC_MoveRelative1.Execute := TRUE;
		nSeqState := STATE_RELIEF_WAIT_MOVE;

	STATE_RELIEF_WAIT_MOVE:
		IF fbMC_MoveRelative1.Done THEN
			fbMC_MoveRelative1.Execute := FALSE;
			bError := TRUE;
			nErrorCode := ERROR_RELIEF_COMPLETED;
			nAxisErrorID := 0;
			nSeqState := STATE_ERROR_LATCHED;
		END_IF
END_CASE

// Saved-position restore is a service operation and is independent of nMode.
IF rtRestorePosition.Q AND nSeqState = STATE_IDLE AND
	NOT bError AND NOT bSafetyError THEN
	IF bExternalBusy THEN
		stMoveCommand.bExecute := FALSE;
		SetError(
			nCode := ERROR_COMMAND_CONFLICT,
			nNativeErrorID := 0,
			bRequestHalt := TRUE);
	ELSIF NOT bPowerState THEN
		stMoveCommand.bExecute := FALSE;
		SetError(
			nCode := ERROR_POWER_UNAVAILABLE,
			nNativeErrorID := 0,
			bRequestHalt := TRUE);
	ELSIF NOT bSavedPositionValid THEN
		stMoveCommand.bExecute := FALSE;
		SetError(
			nCode := ERROR_SAVED_POSITION_UNAVAILABLE,
			nNativeErrorID := 0,
			bRequestHalt := TRUE);
	ELSIF NOT ((stMoveCommand.fRestoreVelocity =
		stMoveCommand.fRestoreVelocity) AND
		ABS(stMoveCommand.fRestoreVelocity) > 0.0 AND
		ABS(stMoveCommand.fRestoreVelocity) < 1.0E300) THEN
		stMoveCommand.bExecute := FALSE;
		SetError(
			nCode := ERROR_INVALID_RUNTIME_VALUE,
			nNativeErrorID := 0,
			bRequestHalt := TRUE);
	ELSE
		fTestStartPos := fActPosition;
		nSystemStatus := STATUS_BASIC_MOVE;
		nLoadDirection := 0;
		nLastMotionDirection := 0;
		nReliefSourceDirection := 0;
		PreparePositionEndpoint(
			fTargetPosition := fSavedPosition,
			fRate := stMoveCommand.fRestoreVelocity,
			nTargetSyncPoint := SYNC_NONE,
			nTargetSyncCycle := 0,
			nNextState := STATE_RESTORE_COMPLETE);
	END_IF
END_IF

// =========================================================
//                      Mode switcher
// =========================================================

IF NOT bError AND NOT bSafetyError AND
	nSeqState < STATE_ABORT_STOPPING THEN
	IF nSeqState >= STATE_POSITION_PREPARE AND
		nSeqState <= STATE_POSITION_BARRIER THEN
		positionEndpoint();
	ELSIF nSeqState >= STATE_FORCE_PREPARE AND
		nSeqState <= STATE_FORCE_HOLD THEN
		forceEndpoint();
	ELSIF nSeqState = STATE_RESTORE_COMPLETE THEN
		testSequence();
	ELSE
		CASE stMoveCommand.nMode OF
			1: mode1();
			2: mode2();
			3: testSequence();
		ELSE
			IF stMoveCommand.bExecute THEN
				stMoveCommand.bExecute := FALSE;
				bError := TRUE;
				nErrorCode := ERROR_UNSUPPORTED_MODE;
			END_IF
		END_CASE
	END_IF
END_IF

// =========================================================
//                      Motion calls
// =========================================================

fbMC_MoveRelative1(
	Axis := Axis,
	Distance := fTargetDist1,
	Velocity := fTargetVel1,
	BufferMode := MC_Aborting);

fbMC_MoveVelocity(
	Axis := Axis,
	Execute := bExecuteVelMove,
	Velocity := ABS(fCmdVelocity),
	Direction := mcDirection,
	BufferMode := MC_Aborting);

IF Axis.Status.PositiveDirection THEN
	nLastMotionDirection := 1;
ELSIF Axis.Status.NegativeDirection THEN
	nLastMotionDirection := -1;
END_IF

// =========================================================
//                         Outputs
// =========================================================

IF nSeqState = STATE_IDLE THEN
	nSystemStatus := STATUS_IDLE;
ELSIF nSeqState >= STATE_ABORT_STOPPING THEN
	nSystemStatus := STATUS_STOPPING;
END_IF

// Expose a newly entered relief state in this scan
bPeerAbortRequest := nSeqState >= STATE_RELIEF_WAIT_STOP AND
	nSeqState <= STATE_RELIEF_WAIT_MOVE;

bBusy := nSeqState > STATE_IDLE AND
	nSeqState <> STATE_ERROR_LATCHED;

IF bOperationCompleted THEN
	nOperationCounter := nOperationCounter + 1;
	bOperationCompleted := FALSE;
END_IF

METHOD ClearActiveCommand

fbMC_MoveRelative1.Execute := FALSE;
bExecuteVelMove := FALSE;
bSinglePrimaryActive := FALSE;
bForceEndpointReady := FALSE;
nSyncPoint := SYNC_NONE;
nSyncCycle := 0;
END_METHOD

ACTION forceEndpoint:

CASE nSeqState OF
	STATE_FORCE_PREPARE:
		bExecuteVelMove := FALSE;
		fForceHoldElapsed := 0.0;
		bForceEndpointReady := FALSE;
		nSyncPoint := SYNC_NONE;
		nSyncCycle := 0;
		fEndpointStartError := fEndpointTargetForce - fForce;
		nVelocityState := 0;
		fCmdVelocity := ABS(fEndpointRate);
		IF fEndpointStartError * INT_TO_LREAL(FORCE_POLARITY) >= 0.0 THEN
			mcDirection := MC_Positive_Direction;
			nLoadDirection := 1;
			nLastMotionDirection := 1;
		ELSE
			mcDirection := MC_Negative_Direction;
			nLoadDirection := -1;
			nLastMotionDirection := -1;
		END_IF
		IF ABS(fEndpointStartError) <= fEndpointTolerance THEN
			stateHalt := TRUE;
			nVelocityState := 3;
			nSeqState := STATE_FORCE_WAIT_STOP;
		ELSE
			nSeqState := STATE_FORCE_EXECUTE;
		END_IF

	STATE_FORCE_EXECUTE: // Trigger constant-speed force approach.
		bExecuteVelMove := TRUE;
		nVelocityState := 1;
		nSeqState := STATE_FORCE_WAIT_TOLERANCE;

	STATE_FORCE_WAIT_TOLERANCE:
		fEndpointCurrentError := fEndpointTargetForce - fForce;
		IF ABS(fEndpointCurrentError) <= fEndpointTolerance OR
			(fEndpointStartError > 0.0 AND fEndpointCurrentError <= 0.0) OR
			(fEndpointStartError < 0.0 AND fEndpointCurrentError >= 0.0) THEN
			bExecuteVelMove := FALSE;
			stateHalt := TRUE;
			nVelocityState := 3;
			nSeqState := STATE_FORCE_WAIT_STOP;
		END_IF

	STATE_FORCE_WAIT_STOP:
		IF bHaltDone THEN
			stateHalt := FALSE;
			nVelocityState := 4;
			nSeqState := STATE_FORCE_HOLD;
		END_IF

	STATE_FORCE_HOLD: // Hold/regulate while synchronized peer catches up.
		IF bForceEndpointReady AND bSyncRelease THEN
			bForceEndpointReady := FALSE;
			nSyncPoint := SYNC_NONE;
			nSyncCycle := 0;
			nEndpointSyncPoint := SYNC_NONE;
			nSeqState := nAfterEndpointState;
		ELSE
			fForceError := fEndpointTargetForce - fForce;

			IF ABS(fForceError) <= fEndpointTolerance THEN
				bExecuteVelMove := FALSE;

				IF nVelocityState <> 3 AND nVelocityState <> 4 THEN
					stateHalt := TRUE;
					nVelocityState := 3;
				ELSIF nVelocityState = 3 AND bHaltDone THEN
					stateHalt := FALSE;
					nVelocityState := 4;
				END_IF

				IF nVelocityState = 4 AND NOT bForceEndpointReady THEN
					fForceHoldElapsed := fForceHoldElapsed + CYCLE_TIME;
					IF fForceHoldElapsed >= fEndpointHoldTime THEN
						IF bSyncEnabled AND
							nEndpointSyncPoint <> SYNC_NONE THEN
							bForceEndpointReady := TRUE;
							nSyncPoint := nEndpointSyncPoint;
							nSyncCycle := nEndpointSyncCycle;
						ELSE
							nSeqState := nAfterEndpointState;
						END_IF
					END_IF
				END_IF
			ELSIF nVelocityState = 3 THEN
				IF bHaltDone THEN
					stateHalt := FALSE;
					nVelocityState := 4;
				END_IF
			ELSIF nVelocityState = 4 THEN
				// Keep elapsed hold time, but withdraw readiness while correcting.
				bForceEndpointReady := FALSE;
				nSyncPoint := SYNC_NONE;
				nSyncCycle := 0;
				fEndpointStartError := fForceError;
				fCmdVelocity := ABS(fEndpointRate);
				IF fForceError * INT_TO_LREAL(FORCE_POLARITY) >= 0.0 THEN
					mcDirection := MC_Positive_Direction;
					nLoadDirection := 1;
					nLastMotionDirection := 1;
				ELSE
					mcDirection := MC_Negative_Direction;
					nLoadDirection := -1;
					nLastMotionDirection := -1;
				END_IF
				nVelocityState := 0;
				nSeqState := STATE_FORCE_EXECUTE;
			END_IF
		END_IF
END_CASE
END_ACTION

ACTION mode1:

// =========================================================
//                  Mode 1: Single relative move
// =========================================================

CASE nSeqState OF
	STATE_IDLE:
		fbMC_MoveRelative1.Execute := FALSE;
		IF stMoveCommand.bExecute THEN
			stMoveCommand.bExecute := FALSE;
			nSystemStatus := STATUS_BASIC_MOVE;
			fTargetDist1 := stMoveCommand.fMoveDistance;
			fTargetVel1 := ABS(stMoveCommand.fMoveVelocity);
			nLoadDirection := 0;
			nReliefSourceDirection := 0;
			IF fTargetDist1 > POSITION_EPSILON THEN
				nLastMotionDirection := 1;
			ELSIF fTargetDist1 < -POSITION_EPSILON THEN
				nLastMotionDirection := -1;
			END_IF
			nSeqState := STATE_MODE_START;
		END_IF

	STATE_MODE_START:
		IF ABS(fTargetDist1) <= POSITION_EPSILON THEN
			bOperationCompleted := TRUE;
			nSeqState := STATE_IDLE;
		ELSE
			fbMC_MoveRelative1.Execute := TRUE;
			nSeqState := STATE_MODE_RUN;
		END_IF

	STATE_MODE_RUN:
		IF fbMC_MoveRelative1.Done THEN
			fbMC_MoveRelative1.Execute := FALSE;
			bOperationCompleted := TRUE;
			nSeqState := STATE_IDLE;
		END_IF
END_CASE
END_ACTION

ACTION mode2:


// =========================================================
//                  Mode 2: Constant Force
// =========================================================
// One PI-regulated target force for one duration.

CASE nSeqState OF
	STATE_IDLE: // Wait for command
		bExecuteVelMove := FALSE;
		fCmdVelocity := 0.0;
		fForceErrorIntegral := 0.0;
		fLastSentVelocity := 0.0;
		IF stMoveCommand.bExecute THEN
			stMoveCommand.bExecute := FALSE;
			nSystemStatus := STATUS_FORCE_MODE;
			nVelocityState := 0;
			nLoadDirection := 0;
			nLastMotionDirection := 0;
			nReliefSourceDirection := 0;
			nSeqState := STATE_MODE_START;
		END_IF

	STATE_MODE_START: // Initialize the single force/time command.
		fTargetForce := stMoveCommand.fTargetForce;
		fForceErrorIntegral := 0.0;
		fMode2HoldElapsed := 0.0;
		fLastSentVelocity := 0.0;
		nVelocityUpdateCounter := VELOCITY_UPDATE_CYCLES;
		nSeqState := STATE_MODE_RUN;

	STATE_MODE_RUN: // Force Regulation Loop (PI Regulator)
		fForceError := fTargetForce - fForce;
		
		fForceErrorIntegral := fForceErrorIntegral + (fForceError * CYCLE_TIME);
		fForceErrorIntegral := LIMIT(-stSettings.fIntegralLimit, fForceErrorIntegral, stSettings.fIntegralLimit);
		
		// Apply the fixed machine force polarity to the PI output.
		fCmdVelocity := ((fForceError * stSettings.fKp) +
			(fForceErrorIntegral * stSettings.fKi)) *
			INT_TO_LREAL(FORCE_POLARITY);
		fCmdVelocity := LIMIT(-stSettings.fMaxVelocity, fCmdVelocity, stSettings.fMaxVelocity);
		
		nVelocityUpdateCounter := nVelocityUpdateCounter + 1;

		IF ABS(fForceError) <= stSettings.fForceTolerance THEN
			// Stop in the force deadband without powering the axis off.
			bExecuteVelMove := FALSE;
			IF nVelocityState <> 3 AND nVelocityState <> 4 THEN
				stateHalt := TRUE;
				nVelocityState := 3;
			ELSIF nVelocityState = 3 AND bHaltDone THEN
				stateHalt := FALSE;
				nVelocityState := 4;
			END_IF
		ELSIF nVelocityState = 3 THEN
			IF bHaltDone THEN
				stateHalt := FALSE;
				nVelocityState := 0;
			END_IF
		ELSIF nVelocityState = 4 THEN
			// The axis is stopped and the force left the deadband.
			nVelocityState := 0;
		ELSIF nVelocityState = 2 THEN
			fCmdVelocity := fPendingVelocity;
			mcDirection := mcPendingDirection;
			bExecuteVelMove := TRUE;
			fLastSentVelocity := fCmdVelocity;
			nVelocityUpdateCounter := 0;
			nVelocityState := 1;
		ELSE
			IF fCmdVelocity >= 0.0 THEN
				mcPendingDirection := MC_Positive_Direction;
			ELSE
				mcPendingDirection := MC_Negative_Direction;
			END_IF
			fPendingVelocity := ABS(fCmdVelocity);

			IF nVelocityState = 0 THEN
				fCmdVelocity := fPendingVelocity;
				mcDirection := mcPendingDirection;
				bExecuteVelMove := TRUE;
				fLastSentVelocity := fCmdVelocity;
				nVelocityUpdateCounter := 0;
				nVelocityState := 1;
			ELSIF nVelocityUpdateCounter >= VELOCITY_UPDATE_CYCLES AND
				(ABS(fPendingVelocity - fLastSentVelocity) >= VELOCITY_UPDATE_DELTA OR
				 mcPendingDirection <> mcDirection) THEN
				bExecuteVelMove := FALSE;
				nVelocityState := 2;
			END_IF
		END_IF
		
		// Count only time spent stopped inside the force tolerance. Leaving the
		// deadband pauses this accumulated time; re-entry resumes it.
		IF ABS(fForceError) <= stSettings.fForceTolerance AND
			nVelocityState = 4 THEN
			fMode2HoldElapsed := fMode2HoldElapsed + CYCLE_TIME;
			IF fMode2HoldElapsed >= stMoveCommand.fForceDuration THEN
				bExecuteVelMove := FALSE;
				stateHalt := FALSE;
				nVelocityState := 0;
				bOperationCompleted := TRUE;
				nSeqState := STATE_IDLE;
			END_IF
		END_IF
END_CASE
END_ACTION

ACTION positionEndpoint:

CASE nSeqState OF
	STATE_POSITION_PREPARE:
		fbMC_MoveRelative1.Execute := FALSE;
		IF ABS(fTargetDist1) <= POSITION_EPSILON THEN
			IF bSyncEnabled AND nEndpointSyncPoint <> SYNC_NONE THEN
				nSyncPoint := nEndpointSyncPoint;
				nSyncCycle := nEndpointSyncCycle;
				nSeqState := STATE_POSITION_BARRIER;
			ELSE
				nSeqState := nAfterEndpointState;
			END_IF
		ELSE
			IF fTargetDist1 > 0.0 THEN
				nLastMotionDirection := 1;
			ELSE
				nLastMotionDirection := -1;
			END_IF
			nSeqState := STATE_POSITION_EXECUTE;
		END_IF

	STATE_POSITION_EXECUTE: // One scan with Execute low before reuse.
		fbMC_MoveRelative1.Execute := TRUE;
		nSeqState := STATE_POSITION_WAIT;

	STATE_POSITION_WAIT:
		IF fbMC_MoveRelative1.Done THEN
			fbMC_MoveRelative1.Execute := FALSE;
			IF bSyncEnabled AND nEndpointSyncPoint <> SYNC_NONE THEN
				nSyncPoint := nEndpointSyncPoint;
				nSyncCycle := nEndpointSyncCycle;
				nSeqState := STATE_POSITION_BARRIER;
			ELSE
				nSeqState := nAfterEndpointState;
			END_IF
		END_IF

	STATE_POSITION_BARRIER: // Powered NC loop holds while peer catches up.
		nSyncPoint := nEndpointSyncPoint;
		nSyncCycle := nEndpointSyncCycle;
		IF NOT bSyncEnabled OR bSyncRelease THEN
			nSyncPoint := SYNC_NONE;
			nSyncCycle := 0;
			nEndpointSyncPoint := SYNC_NONE;
			nSeqState := nAfterEndpointState;
		END_IF
END_CASE
END_ACTION

METHOD PrepareForceEndpoint
VAR_INPUT
	fTargetForceValue : LREAL;
	fRate             : LREAL;
	fTolerance        : LREAL;
	fHoldTime         : LREAL;
	nTargetSyncPoint  : BYTE;
	nTargetSyncCycle  : INT;
	nNextState        : INT;
END_VAR

fEndpointTargetForce := fTargetForceValue;
fEndpointRate := ABS(fRate);
fEndpointTolerance := fTolerance;
fEndpointHoldTime := fHoldTime;
nEndpointSyncPoint := nTargetSyncPoint;
nEndpointSyncCycle := nTargetSyncCycle;
nAfterEndpointState := nNextState;
nSeqState := STATE_FORCE_PREPARE;
END_METHOD

METHOD PreparePositionEndpoint
VAR_INPUT
	fTargetPosition : LREAL;
	fRate           : LREAL;
	nTargetSyncPoint: BYTE;
	nTargetSyncCycle: INT;
	nNextState      : INT;
END_VAR

fEndpointTargetPosition := fTargetPosition;
fTargetDist1 := fEndpointTargetPosition - fActPosition;
fTargetVel1 := ABS(fRate);
nEndpointSyncPoint := nTargetSyncPoint;
nEndpointSyncCycle := nTargetSyncCycle;
nAfterEndpointState := nNextState;
nSeqState := STATE_POSITION_PREPARE;
END_METHOD

METHOD SetError
VAR_INPUT
	nCode          : UDINT;
	nNativeErrorID : UDINT;
	bRequestHalt   : BOOL;
END_VAR

bError := TRUE;
nErrorCode := nCode;
nAxisErrorID := nNativeErrorID;
ClearActiveCommand();
IF bRequestHalt THEN
	stateHalt := TRUE;
	nSeqState := STATE_ERROR_STOPPING;
ELSE
	stateHalt := FALSE;
	nSeqState := STATE_ERROR_LATCHED;
END_IF
END_METHOD

ACTION testSequence:

// Shared pre-test, main-test and post-test sequence for mode 3.
// All stored coordinates are references only; every position command is relative.

// Criterion 2 ends a single test immediately when its signed level is crossed.
IF bSinglePrimaryActive AND stMoveCommand.nStop2Mode > 0 THEN
	bSingleStopReached := FALSE;
	IF stMoveCommand.nStop2Mode = 1 THEN
		fStop2CurrentError := fStop2TargetPosition - fActPosition;
		IF ABS(fStop2CurrentError) <= POSITION_EPSILON OR
			(fStop2StartError > 0.0 AND fStop2CurrentError <= 0.0) OR
			(fStop2StartError < 0.0 AND fStop2CurrentError >= 0.0) THEN
			bSingleStopReached := TRUE;
		END_IF
	ELSIF stMoveCommand.nStop2Mode = 2 THEN
		fStop2CurrentError := stMoveCommand.fStop2Value - fForce;
		IF ABS(fStop2CurrentError) <= stMoveCommand.fSingleForceTolerance OR
			(fStop2StartError > 0.0 AND fStop2CurrentError <= 0.0) OR
			(fStop2StartError < 0.0 AND fStop2CurrentError >= 0.0) THEN
			bSingleStopReached := TRUE;
		END_IF
	END_IF

	IF bSingleStopReached THEN
		fbMC_MoveRelative1.Execute := FALSE;
		bExecuteVelMove := FALSE;
		bSinglePrimaryActive := FALSE;
		stateHalt := TRUE;
		nSeqState := STATE_SINGLE_WAIT_STOP;
	END_IF
END_IF

CASE nSeqState OF
	STATE_IDLE: // Start a test. MATLAB keeps command values unchanged while bWorking is TRUE.
		fbMC_MoveRelative1.Execute := FALSE;
		bExecuteVelMove := FALSE;
		stateHalt := FALSE;
		bSinglePrimaryActive := FALSE;
		bForceEndpointReady := FALSE;
		nSyncPoint := SYNC_NONE;
		nSyncCycle := 0;
		nEndpointSyncPoint := SYNC_NONE;
		nEndpointSyncCycle := 0;

		IF stMoveCommand.bExecute THEN
			stMoveCommand.bExecute := FALSE;
			IF stMoveCommand.nCycleCount < 0 OR
				stMoveCommand.nCycleCount > 50 OR
				stMoveCommand.nPreCycleCount < 0 OR
				stMoveCommand.nPreCycleCount > 50 OR
				(stMoveCommand.bPreTestOnly AND NOT stMoveCommand.bIncludePreTest) OR
				NOT ((stMoveCommand.fPreTestForceTolerance = stMoveCommand.fPreTestForceTolerance) AND
					ABS(stMoveCommand.fPreTestForceTolerance) < 1.0E300 AND
					stMoveCommand.fPreTestForceTolerance >= 0.0) OR
				NOT ((stMoveCommand.fPreloadHoldTime = stMoveCommand.fPreloadHoldTime) AND
					ABS(stMoveCommand.fPreloadHoldTime) < 1.0E300 AND
					stMoveCommand.fPreloadHoldTime >= 0.0) OR
				NOT ((stMoveCommand.fPreCycleHoldTime = stMoveCommand.fPreCycleHoldTime) AND
					ABS(stMoveCommand.fPreCycleHoldTime) < 1.0E300 AND
					stMoveCommand.fPreCycleHoldTime >= 0.0) OR
				NOT ((stMoveCommand.fSingleForceTolerance = stMoveCommand.fSingleForceTolerance) AND
					ABS(stMoveCommand.fSingleForceTolerance) < 1.0E300 AND
					stMoveCommand.fSingleForceTolerance >= 0.0) OR
				NOT ((stMoveCommand.fSingleForceHoldTime = stMoveCommand.fSingleForceHoldTime) AND
					ABS(stMoveCommand.fSingleForceHoldTime) < 1.0E300 AND
					stMoveCommand.fSingleForceHoldTime >= 0.0) OR
				NOT ((stMoveCommand.fCyclicForceTolerance = stMoveCommand.fCyclicForceTolerance) AND
					ABS(stMoveCommand.fCyclicForceTolerance) < 1.0E300 AND
					stMoveCommand.fCyclicForceTolerance >= 0.0) OR
				NOT ((stMoveCommand.fCyclicForceHoldTime = stMoveCommand.fCyclicForceHoldTime) AND
					ABS(stMoveCommand.fCyclicForceHoldTime) < 1.0E300 AND
					stMoveCommand.fCyclicForceHoldTime >= 0.0) THEN
				bError := TRUE;
				nErrorCode := ERROR_INVALID_CONFIGURATION;
				stateHalt := TRUE;
				nSeqState := STATE_ERROR_STOPPING;
			ELSE
				fTestStartPos := fActPosition;
				fPreTestFinalPos := fTestStartPos;
				nCurrentCycle := 1;
				nCurrentPreCycle := 1;
				nLoadDirection := 0;
				nLastMotionDirection := 0;
				nReliefSourceDirection := 0;
				nVelocityState := 0;

				IF stMoveCommand.bIncludePreTest THEN
					IF stMoveCommand.bPreloadEnabled THEN
						nSystemStatus := STATUS_PRETENSION;
					ELSE
						nSystemStatus := STATUS_PRETEST_CYCLIC;
					END_IF
					nSeqState := STATE_PRELOAD;
				ELSE
					IF stMoveCommand.nCycleCount > 0 THEN
						nSystemStatus := STATUS_CYCLIC_TEST;
					ELSE
						nSystemStatus := STATUS_SINGLE_TEST;
					END_IF
					nSeqState := STATE_SELECT_MAIN_TEST;
				END_IF
			END_IF
		END_IF

	STATE_PRELOAD: // Optional one-time force preload.
		nCurrentPreCycle := 1;
		IF stMoveCommand.bPreloadEnabled THEN
			nSystemStatus := STATUS_PRETENSION;
			fEndpointTargetForce := stMoveCommand.fPreloadValue;
			fEndpointRate := ABS(stMoveCommand.fPreTestRate);
			fEndpointTolerance := stMoveCommand.fPreTestForceTolerance;
			fEndpointHoldTime := stMoveCommand.fPreloadHoldTime;
			nEndpointSyncPoint := SYNC_PRETENSION_DONE;
			nEndpointSyncCycle := 0;
			nAfterEndpointState := STATE_CAPTURE_TEST_START;
			nSeqState := STATE_FORCE_PREPARE;
		ELSE
			nSystemStatus := STATUS_PRETEST_CYCLIC;
			nSeqState := STATE_PRE_CYCLE_LOAD;
		END_IF

	STATE_CAPTURE_TEST_START: // Capture post-pretension test start.
		fTestStartPos := fActPosition;
		IF stMoveCommand.nPreCycleCount > 0 THEN
			nSystemStatus := STATUS_PRETEST_CYCLIC;
			nSeqState := STATE_PRE_CYCLE_LOAD;
		ELSE
			nSeqState := STATE_CAPTURE_PRETEST_FINAL;
		END_IF

	STATE_PRE_CYCLE_LOAD: // Pre-conditioning force-load endpoint.
		nSystemStatus := STATUS_PRETEST_CYCLIC;
		IF nCurrentPreCycle > stMoveCommand.nPreCycleCount THEN
			nSeqState := STATE_PRETEST_BARRIER;
		ELSE
			fEndpointTargetForce := stMoveCommand.fPreCycleLoadValue;
			fEndpointRate := ABS(stMoveCommand.fPreTestRate);
			fEndpointTolerance := stMoveCommand.fPreTestForceTolerance;
			fEndpointHoldTime := stMoveCommand.fPreCycleHoldTime;
			nEndpointSyncPoint := SYNC_LOAD_DONE;
			nEndpointSyncCycle := nCurrentPreCycle;
			nAfterEndpointState := STATE_PRE_CYCLE_UNLOAD;
			nSeqState := STATE_FORCE_PREPARE;
		END_IF

	STATE_PRE_CYCLE_UNLOAD: // Force unload or return to test start.
		nSystemStatus := STATUS_PRETEST_CYCLIC;
		IF stMoveCommand.bPreUnloadToStart THEN
			fEndpointTargetPosition := fTestStartPos;
			fTargetDist1 := fEndpointTargetPosition - fActPosition;
			fTargetVel1 := ABS(stMoveCommand.fPreTestRate);
			IF nCurrentPreCycle = stMoveCommand.nPreCycleCount THEN
				nEndpointSyncPoint := SYNC_PRETEST_DONE;
				nAfterEndpointState := STATE_CAPTURE_PRETEST_FINAL;
			ELSE
				nEndpointSyncPoint := SYNC_UNLOAD_DONE;
				nAfterEndpointState := STATE_PRE_CYCLE_NEXT;
			END_IF
			nEndpointSyncCycle := nCurrentPreCycle;
			nSeqState := STATE_POSITION_PREPARE;
		ELSE
			fEndpointTargetForce := stMoveCommand.fPreUnloadValue;
			fEndpointRate := ABS(stMoveCommand.fPreTestRate);
			fEndpointTolerance := stMoveCommand.fPreTestForceTolerance;
			fEndpointHoldTime := stMoveCommand.fPreCycleHoldTime;
			IF nCurrentPreCycle = stMoveCommand.nPreCycleCount THEN
				nEndpointSyncPoint := SYNC_PRETEST_DONE;
				nAfterEndpointState := STATE_CAPTURE_PRETEST_FINAL;
			ELSE
				nEndpointSyncPoint := SYNC_UNLOAD_DONE;
				nAfterEndpointState := STATE_PRE_CYCLE_NEXT;
			END_IF
			nEndpointSyncCycle := nCurrentPreCycle;
			nSeqState := STATE_FORCE_PREPARE;
		END_IF

	STATE_PRE_CYCLE_NEXT:
		nCurrentPreCycle := nCurrentPreCycle + 1;
		nSeqState := STATE_PRE_CYCLE_LOAD;

	STATE_CAPTURE_PRETEST_FINAL: // Final pre-test endpoint passed its barrier.
		fPreTestFinalPos := fActPosition;
		IF stMoveCommand.bPreTestOnly THEN
			nSystemStatus := STATUS_POSTTEST;
			nSeqState := STATE_POSTTEST_SELECT;
		ELSE
			IF stMoveCommand.nCycleCount > 0 THEN
				nSystemStatus := STATUS_CYCLIC_TEST;
			ELSE
				nSystemStatus := STATUS_SINGLE_TEST;
			END_IF
			nSeqState := STATE_SELECT_MAIN_TEST;
		END_IF

	STATE_PRETEST_BARRIER: // No final endpoint; explicit pre-test barrier.
		nSystemStatus := STATUS_PRETEST_CYCLIC;
		nSyncPoint := SYNC_PRETEST_DONE;
		nSyncCycle := 0;
		IF NOT bSyncEnabled OR bSyncRelease THEN
			nSyncPoint := SYNC_NONE;
			fPreTestFinalPos := fActPosition;
			IF stMoveCommand.bPreTestOnly THEN
				nSystemStatus := STATUS_POSTTEST;
				nSeqState := STATE_POSTTEST_SELECT;
			ELSE
				IF stMoveCommand.nCycleCount > 0 THEN
					nSystemStatus := STATUS_CYCLIC_TEST;
				ELSE
					nSystemStatus := STATUS_SINGLE_TEST;
				END_IF
				nSeqState := STATE_SELECT_MAIN_TEST;
			END_IF
		END_IF

	STATE_SELECT_MAIN_TEST: // Positive cycle count selects cyclic.
		IF stMoveCommand.nCycleCount > 0 THEN
			nSystemStatus := STATUS_CYCLIC_TEST;
			nSeqState := STATE_CYCLIC_LOAD;
		ELSE
			nSystemStatus := STATUS_SINGLE_TEST;
			nSeqState := STATE_SINGLE_START;
		END_IF

	// -----------------------------------------------------
	// Mode 3: cyclic load endpoint followed by unload endpoint
	// -----------------------------------------------------
	STATE_CYCLIC_LOAD:
		nSystemStatus := STATUS_CYCLIC_TEST;
		IF nCurrentCycle > stMoveCommand.nCycleCount THEN
			nSeqState := STATE_POSTTEST_SELECT;
		ELSIF stMoveCommand.nLoadMode = 1 THEN
			fEndpointTargetPosition := fPreTestFinalPos +
				stMoveCommand.fLoadValues[nCurrentCycle];
			fTargetDist1 := fEndpointTargetPosition - fActPosition;
			fTargetVel1 := ABS(stMoveCommand.fTestRate);
			IF fTargetDist1 > POSITION_EPSILON THEN
				nLoadDirection := 1;
			ELSIF fTargetDist1 < -POSITION_EPSILON THEN
				nLoadDirection := -1;
			END_IF
			nEndpointSyncPoint := SYNC_LOAD_DONE;
			nEndpointSyncCycle := nCurrentCycle;
			nAfterEndpointState := STATE_CYCLIC_UNLOAD;
			nSeqState := STATE_POSITION_PREPARE;
		ELSIF stMoveCommand.nLoadMode = 2 THEN
			fEndpointTargetForce := stMoveCommand.fLoadValues[nCurrentCycle];
			fEndpointRate := ABS(stMoveCommand.fTestRate);
			fEndpointTolerance := stMoveCommand.fCyclicForceTolerance;
			fEndpointHoldTime := stMoveCommand.fCyclicForceHoldTime;
			nEndpointSyncPoint := SYNC_LOAD_DONE;
			nEndpointSyncCycle := nCurrentCycle;
			nAfterEndpointState := STATE_CYCLIC_UNLOAD;
			nSeqState := STATE_FORCE_PREPARE;
		ELSE
			bError := TRUE;
			nErrorCode := ERROR_UNSUPPORTED_ENDPOINT;
			stateHalt := TRUE;
			nSeqState := STATE_ERROR_STOPPING;
		END_IF

	STATE_CYCLIC_UNLOAD:
		nSystemStatus := STATUS_CYCLIC_TEST;
		IF stMoveCommand.nUnloadMode = 1 THEN
			fEndpointTargetPosition := fPreTestFinalPos +
				stMoveCommand.fUnloadValues[nCurrentCycle];
			fTargetDist1 := fEndpointTargetPosition - fActPosition;
			fTargetVel1 := ABS(stMoveCommand.fTestRate);
			IF nCurrentCycle = stMoveCommand.nCycleCount THEN
				nEndpointSyncPoint := SYNC_MAIN_DONE;
				nAfterEndpointState := STATE_CYCLIC_COMPLETE;
			ELSE
				nEndpointSyncPoint := SYNC_UNLOAD_DONE;
				nAfterEndpointState := STATE_CYCLIC_NEXT;
			END_IF
			nEndpointSyncCycle := nCurrentCycle;
			nSeqState := STATE_POSITION_PREPARE;
		ELSIF stMoveCommand.nUnloadMode = 2 THEN
			fEndpointTargetForce := stMoveCommand.fUnloadValues[nCurrentCycle];
			fEndpointRate := ABS(stMoveCommand.fTestRate);
			fEndpointTolerance := stMoveCommand.fCyclicForceTolerance;
			fEndpointHoldTime := stMoveCommand.fCyclicForceHoldTime;
			IF nCurrentCycle = stMoveCommand.nCycleCount THEN
				nEndpointSyncPoint := SYNC_MAIN_DONE;
				nAfterEndpointState := STATE_CYCLIC_COMPLETE;
			ELSE
				nEndpointSyncPoint := SYNC_UNLOAD_DONE;
				nAfterEndpointState := STATE_CYCLIC_NEXT;
			END_IF
			nEndpointSyncCycle := nCurrentCycle;
			nSeqState := STATE_FORCE_PREPARE;
		ELSE
			bError := TRUE;
			nErrorCode := ERROR_UNSUPPORTED_ENDPOINT;
			stateHalt := TRUE;
			nSeqState := STATE_ERROR_STOPPING;
		END_IF

	STATE_CYCLIC_NEXT:
		nCurrentCycle := nCurrentCycle + 1;
		nSeqState := STATE_CYCLIC_LOAD;

	STATE_CYCLIC_COMPLETE: // Final unload also serves as main barrier.
		nCurrentCycle := nCurrentCycle + 1;
		nSeqState := STATE_POSTTEST_SELECT;

	// -----------------------------------------------------
	// Mode 3 single test: criterion 1 is the primary endpoint
	// -----------------------------------------------------
	STATE_SINGLE_START:
		nSystemStatus := STATUS_SINGLE_TEST;
		bSingleStopReached := FALSE;
		bSinglePrimaryActive := TRUE;

		IF stMoveCommand.nStop2Mode = 1 THEN
			fStop2TargetPosition := fPreTestFinalPos + stMoveCommand.fStop2Value;
			fStop2StartError := fStop2TargetPosition - fActPosition;
		ELSIF stMoveCommand.nStop2Mode = 2 THEN
			fStop2StartError := stMoveCommand.fStop2Value - fForce;
		END_IF

		IF stMoveCommand.nStop1Mode = 1 THEN
			fEndpointTargetPosition := fPreTestFinalPos + stMoveCommand.fStop1Value;
			fTargetDist1 := fEndpointTargetPosition - fActPosition;
			fTargetVel1 := ABS(stMoveCommand.fTestRate);
			IF fTargetDist1 > POSITION_EPSILON THEN
				nLoadDirection := 1;
			ELSIF fTargetDist1 < -POSITION_EPSILON THEN
				nLoadDirection := -1;
			END_IF
			nEndpointSyncPoint := SYNC_MAIN_DONE;
			nEndpointSyncCycle := 0;
			nAfterEndpointState := STATE_POSTTEST_SELECT;
			nSeqState := STATE_POSITION_PREPARE;
		ELSIF stMoveCommand.nStop1Mode = 2 THEN
			fEndpointTargetForce := stMoveCommand.fStop1Value;
			fEndpointRate := ABS(stMoveCommand.fTestRate);
			fEndpointTolerance := stMoveCommand.fSingleForceTolerance;
			fEndpointHoldTime := stMoveCommand.fSingleForceHoldTime;
			nEndpointSyncPoint := SYNC_MAIN_DONE;
			nEndpointSyncCycle := 0;
			nAfterEndpointState := STATE_POSTTEST_SELECT;
			nSeqState := STATE_FORCE_PREPARE;
		ELSE
			bSinglePrimaryActive := FALSE;
			bError := TRUE;
			nErrorCode := ERROR_UNSUPPORTED_ENDPOINT;
			stateHalt := TRUE;
			nSeqState := STATE_ERROR_STOPPING;
		END_IF

	STATE_SINGLE_WAIT_STOP: // Optional OR criterion stopped primary.
		IF bHaltDone THEN
			stateHalt := FALSE;
			nVelocityState := 0;
			nSeqState := STATE_SECONDARY_BARRIER;
		END_IF

	STATE_SECONDARY_BARRIER: // Secondary criterion ended test early.
		nSystemStatus := STATUS_SINGLE_TEST;
		nSyncPoint := SYNC_MAIN_DONE;
		nSyncCycle := 0;
		IF NOT bSyncEnabled OR bSyncRelease THEN
			nSyncPoint := SYNC_NONE;
			nSeqState := STATE_POSTTEST_SELECT;
		END_IF

	// -----------------------------------------------------
	// Post-test; reached only after normal main-test completion
	// -----------------------------------------------------
	STATE_POSTTEST_SELECT:
		nSystemStatus := STATUS_POSTTEST;
		bSinglePrimaryActive := FALSE;
		CASE stMoveCommand.nPostTestMode OF
			0: // Stay at the current position.
				fbMC_MoveRelative1.Execute := FALSE;
				bExecuteVelMove := FALSE;
				stateHalt := TRUE;
				nSeqState := STATE_POSTTEST_WAIT_STOP;

			1: // Return to the separately saved coordinate.
				IF bSavedPositionValid THEN
					PreparePositionEndpoint(
						fTargetPosition := fSavedPosition,
						fRate := stMoveCommand.fTestRate,
						nTargetSyncPoint := SYNC_POSTTEST_DONE,
						nTargetSyncCycle := 0,
						nNextState := STATE_OPERATION_COMPLETE);
				ELSE
					stMoveCommand.bExecute := FALSE;
					SetError(
						nCode := ERROR_SAVED_POSITION_UNAVAILABLE,
						nNativeErrorID := 0,
						bRequestHalt := TRUE);
				END_IF

			2: // Return to the test-start position captured after pretension.
				PreparePositionEndpoint(
					fTargetPosition := fTestStartPos,
					fRate := stMoveCommand.fTestRate,
					nTargetSyncPoint := SYNC_POSTTEST_DONE,
					nTargetSyncCycle := 0,
					nNextState := STATE_OPERATION_COMPLETE);

			3: // Return to the actual position reached after pre-test.
				PreparePositionEndpoint(
					fTargetPosition := fPreTestFinalPos,
					fRate := stMoveCommand.fTestRate,
					nTargetSyncPoint := SYNC_POSTTEST_DONE,
					nTargetSyncCycle := 0,
					nNextState := STATE_OPERATION_COMPLETE);

			4: // Release to signed zero force without a hold period.
				PrepareForceEndpoint(
					fTargetForceValue := 0.0,
					fRate := stMoveCommand.fTestRate,
					fTolerance := stSettings.fForceTolerance,
					fHoldTime := 0.0,
					nTargetSyncPoint := SYNC_POSTTEST_DONE,
					nTargetSyncCycle := 0,
					nNextState := STATE_OPERATION_COMPLETE);

		ELSE
			stMoveCommand.bExecute := FALSE;
			SetError(
				nCode := ERROR_UNSUPPORTED_POST_ACTION,
				nNativeErrorID := 0,
				bRequestHalt := TRUE);
		END_CASE

	STATE_POSTTEST_WAIT_STOP:
		IF bHaltDone THEN
			stateHalt := FALSE;
			nSeqState := STATE_POSTTEST_BARRIER;
		END_IF

	STATE_POSTTEST_BARRIER: // Stay mode participates in post-test barrier.
		nSystemStatus := STATUS_POSTTEST;
		nSyncPoint := SYNC_POSTTEST_DONE;
		nSyncCycle := 0;
		IF NOT bSyncEnabled OR bSyncRelease THEN
			nSyncPoint := SYNC_NONE;
			nSeqState := STATE_OPERATION_COMPLETE;
		END_IF

	STATE_OPERATION_COMPLETE:
		nSystemStatus := STATUS_IDLE;
		nSyncPoint := SYNC_NONE;
		nSyncCycle := 0;
		bOperationCompleted := TRUE;
		nSeqState := STATE_IDLE;

	STATE_RESTORE_COMPLETE: // Standalone saved-position restore completed.
		nSystemStatus := STATUS_IDLE;
		bOperationCompleted := TRUE;
		nSeqState := STATE_IDLE;
END_CASE
END_ACTION

END_FUNCTION_BLOCK
